Staubli VAL3: setItem.pgx

public program setItem(InstrItem& x_sItem[] (dimensions=1), num& x_nIndex[] (dimensions=1))
begin
  // set IT
  pEdit.iEvent[x_nIndex]=x_sItem
end
